TYPE "PPrf_SetUp_Man"
VERSION : 0.1
// Block: PPrf_SetUp_Man
   STRUCT
      X : Array[1..SET_UP_MAN_ADJUST_MAX] of Real;
      Y : Array[1..SETUP_MAN_OP_WITH_CODE_QTY] of Int;
   END_STRUCT;

END_TYPE
